Fanuc KAREL source: ka00092.KL

PROGRAM KA00092
%NOLOCKGROUP
VAR
SRC : JOINTPOS9
DST : JOINTPOS9
BEGIN
DST=SRC
END KA00092
